// TIA Portal V16 export
// export: Created 2021-03-05T14:22:13.474108Z, ExportSetting WithDefaults, DisplayName Totally Integrated Automation Portal, DisplayVersion V16, DisplayName TIA Portal Version Control Interface, DisplayVersion V16, DisplayName TIA Portal Openness, DisplayVersion V16, DisplayName SINAMICS Startdrive Advanced, DisplayVersion V16, DisplayName SINAMICS Startdrive G130, G150, S120, S150, SINAMICS MV, S210, DisplayVersion V16, DisplayName SINAMICS Startdrive G110M, G120, G120C, G120D, G120P, DisplayVersion V16, DisplayName STEP 7 Professional, DisplayVersion V16, DisplayName STEP 7 Safety, DisplayVersion V16, DisplayName WinCC Professional, DisplayVersion V16
VAR_GLOBAL   // PLC tag table "Default tag table"
   Clock_Byte AT %MB0 : Byte;
   Clock_10Hz AT %M0.0 : Bool;
   Clock_5Hz AT %M0.1 : Bool;
   "Clock_2.5Hz" AT %M0.2 : Bool;
   Clock_2Hz AT %M0.3 : Bool;
   "Clock_1.25Hz" AT %M0.4 : Bool;
   Clock_1Hz AT %M0.5 : Bool;
   "Clock_0.625Hz" AT %M0.6 : Bool;
   "Clock_0.5Hz" AT %M0.7 : Bool;
   System_Byte AT %MB1 : Byte;
   FirstScan AT %M1.0 : Bool;
   DiagStatusUpdate AT %M1.1 : Bool;
   AlwaysTRUE AT %M1.2 : Bool;
   AlwaysFALSE AT %M1.3 : Bool;
   Rack_1_Reservoir_Level AT %IW11 : Int;
   Rack_2_Reservoir_Level AT %IW13 : Int;
   Rack_3_Reservoir_Level AT %IW15 : Int;
   Rack_4_Reservoir_Level AT %IW17 : Int;
   Rack_1_Shelf_1_Fill AT %Q0.0 : Bool;
   Rack_1_Shelf_1_Drain AT %Q0.1 : Bool;
   Rack_1_Shelf_2_Fill AT %Q0.2 : Bool;
   Rack_1_Shelf_2_Drain AT %Q0.3 : Bool;
   Rack_1_Shelf_3_Fill AT %Q0.4 : Bool;
   Rack_1_Shelf_3_Drain AT %Q0.5 : Bool;
   Rack_1_Shelf_4_Fill AT %Q0.6 : Bool;
   Rack_1_Shelf_4_Drain AT %Q0.7 : Bool;
   Rack_1_Shelf_5_Fill AT %Q1.0 : Bool;
   Rack_1_Shelf_5_Drain AT %Q1.1 : Bool;
   Rack_1_Shelf_6_Fill AT %Q1.2 : Bool;
   Rack_1_Shelf_6_Drain AT %Q1.3 : Bool;
   Rack_1_RO AT %Q1.4 : Bool;
   Rack_1_Discharge AT %Q1.5 : Bool;
   Rack_2_Shelf_1_Fill AT %Q1.6 : Bool;
   Rack_2_Shelf_1_Drain AT %Q1.7 : Bool;
   Rack_2_Shelf_2_Fill AT %Q2.0 : Bool;
   Rack_2_Shelf_2_Drain AT %Q2.1 : Bool;
   Rack_2_Shelf_3_Fill AT %Q2.2 : Bool;
   Rack_2_Shelf_3_Drain AT %Q2.3 : Bool;
   Rack_2_Shelf_4_Fill AT %Q2.4 : Bool;
   Rack_2_Shelf_4_Drain AT %Q2.5 : Bool;
   Rack_2_Shelf_5_Fill AT %Q2.6 : Bool;
   Rack_2_Shelf_5_Drain AT %Q2.7 : Bool;
   Rack_2_Shelf_6_Fill AT %Q3.0 : Bool;
   Rack_2_Shelf_6_Drain AT %Q3.1 : Bool;
   Rack_2_RO AT %Q3.2 : Bool;
   Rack_2_Discharge AT %Q3.3 : Bool;
   Rack_3_Shelf_1_Fill AT %Q3.4 : Bool;
   Rack_3_Shelf_1_Drain AT %Q3.5 : Bool;
   Rack_3_Shelf_2_Fill AT %Q3.6 : Bool;
   Rack_3_Shelf_2_Drain AT %Q3.7 : Bool;
   Rack_3_Shelf_3_Fill AT %Q4.0 : Bool;
   Rack_3_Shelf_3_Drain AT %Q4.1 : Bool;
   Rack_3_Shelf_4_Fill AT %Q4.2 : Bool;
   Rack_3_Shelf_4_Drain AT %Q4.3 : Bool;
   Rack_3_Shelf_5_Fill AT %Q4.4 : Bool;
   Rack_3_Shelf_5_Drain AT %Q4.5 : Bool;
   Rack_3_Shelf_6_Fill AT %Q4.6 : Bool;
   Rack_3_Shelf_6_Drain AT %Q4.7 : Bool;
   Rack_3_RO AT %Q5.0 : Bool;
   Rack_3_Discharge AT %Q5.1 : Bool;
   Rack_4_Shelf_1_Fill AT %Q5.2 : Bool;
   Rack_4_Shelf_1_Drain AT %Q5.3 : Bool;
   Rack_4_Shelf_2_Fill AT %Q5.4 : Bool;
   Rack_4_Shelf_2_Drain AT %Q5.5 : Bool;
   Rack_4_Shelf_3_Fill AT %Q5.6 : Bool;
   Rack_4_Shelf_3_Drain AT %Q5.7 : Bool;
   Rack_4_Shelf_4_Fill AT %Q6.0 : Bool;
   Rack_4_Shelf_4_Drain AT %Q6.1 : Bool;
   Rack_4_Shelf_5_Fill AT %Q6.2 : Bool;
   Rack_4_Shelf_5_Drain AT %Q6.3 : Bool;
   Rack_4_Shelf_6_Fill AT %Q6.4 : Bool;
   Rack_4_Shelf_6_Drain AT %Q6.5 : Bool;
   Rack_4_RO AT %Q6.6 : Bool;
   Rack_4_Discharge AT %Q6.7 : Bool;
   DI_Level_SW_R1S1 AT %I0.0 : Bool;
   DI_Level_SW_R1S2 AT %I0.1 : Bool;
   DI_Level_SW_R1S3 AT %I0.2 : Bool;
   DI_Level_SW_R1S4 AT %I0.3 : Bool;
   DI_Level_SW_R1S5 AT %I0.4 : Bool;
   DI_Level_SW_R1S6 AT %I0.5 : Bool;
   DI_Level_SW_R2S1 AT %I0.6 : Bool;
   DI_Level_SW_R2S2 AT %I0.7 : Bool;
   DI_Level_SW_R2S3 AT %I9.0 : Bool;
   DI_Level_SW_R2S4 AT %I9.1 : Bool;
   DI_Level_SW_R2S5 AT %I9.2 : Bool;
   DI_Level_SW_R2S6 AT %I9.3 : Bool;
   DI_Level_SW_R3S1 AT %I9.4 : Bool;
   DI_Level_SW_R3S2 AT %I9.5 : Bool;
   DI_Level_SW_R3S3 AT %I9.6 : Bool;
   DI_Level_SW_R3S4 AT %I9.7 : Bool;
   DI_Level_SW_R3S5 AT %I10.0 : Bool;
   DI_Level_SW_R3S6 AT %I10.1 : Bool;
   DI_Level_SW_R4S1 AT %I10.2 : Bool;
   DI_Level_SW_R4S2 AT %I10.3 : Bool;
   DI_Level_SW_R4S3 AT %I10.4 : Bool;
   DI_Level_SW_R4S4 AT %I10.5 : Bool;
   DI_Level_SW_R4S5 AT %I10.6 : Bool;
   DI_Level_SW_R4S6 AT %I10.7 : Bool;
END_VAR
